// SIMATIC S7-200 SMART project (STEP 7-Micro/WIN SMART), CPU SR20

SYMBOL_TABLE System Symbols
Clock_1s         SM0.5    // Clock pulse that is ON for 0.5 s, OFF for 0.5 s, for a duty cycle time of 1 s.
END_SYMBOL_TABLE

ORGANIZATION_BLOCK MAIN:OB1
TITLE=Program Comments
BEGIN
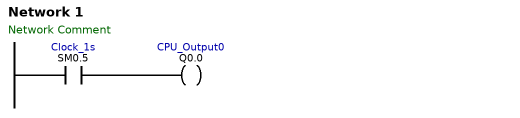
Network 1
// Network Comment
// (network saved uncompiled; LAD cells follow)
// row 0: c0 -| |- Clock_1s:SM0.5  c1 -( ) CPU_Output0:Q0.0
END_ORGANIZATION_BLOCK
